TYPE ST_HW_OutputsSickScanner_CLV690 :
STRUCT
	ConfMessageOut	: ARRAY[0..31] OF BYTE;
	Trigger			: BOOL; // Trigger signal to scanner
END_STRUCT
END_TYPE

(* stored: Version 1.1.0.1, ProductVersion 3.1.4024.4
   DUT ST_HW_OutputsSickScanner_CLV690: Id {0125f6d3-3f3e-4000-9680-de735f4023a0} *)
